GVL_1.Scope_T_Vor_WT_IN :=T_Vor_WT_IN ;
GVL_1.Scope_T_Vor_WT:=T_Vor_WT;
GVL_1.Scope_T_Vor_WT_Visu:=T_Vor_WT_Visu;
GVL_1.Scope_T_nach_WT_IN :=T_nach_WT_IN ;
GVL_1.Scope_T_nach_WT:=T_nach_WT;
GVL_1.Scope_T_nach_WT_Visu:=T_nach_WT_Visu;
GVL_1.Scope_T_HE_Einduesung_Oben_IN :=T_HE_Einduesung_Oben_IN ;
GVL_1.Scope_T_HE_Einduesung_Oben:=T_HE_Einduesung_Oben;
GVL_1.Scope_T_HE_Einduesung_Oben_Visu:=T_HE_Einduesung_Oben_Visu;
GVL_1.Scope_T_HE_Einduesung_Unten_IN :=T_HE_Einduesung_Unten_IN ;
GVL_1.Scope_T_HE_Einduesung_Unten:=T_HE_Einduesung_Unten;
GVL_1.Scope_T_HE_Einduesung_Unten_Visu:=T_HE_Einduesung_Unten_Visu;
GVL_1.Scope_T_Einduesung_Unten_IN :=T_Einduesung_Unten_IN ;
GVL_1.Scope_T_Einduesung_Unten:=T_Einduesung_Unten;
GVL_1.Scope_T_Einduesung_Unten_Visu:=T_Einduesung_Unten_Visu;
GVL_1.Scope_T_Einduesung_Oben_IN :=T_Einduesung_Oben_IN ;
GVL_1.Scope_T_Einduesung_Oben:=T_Einduesung_Oben;
GVL_1.Scope_T_Einduesung_Oben_Visu:=T_Einduesung_Oben_Visu;
GVL_1.Scope_T_Absaugung_Oben_IN :=T_Absaugung_Oben_IN ;
GVL_1.Scope_T_Absaugung_Oben:=T_Absaugung_Oben;
GVL_1.Scope_T_Absaugung_Oben_Visu:=T_Absaugung_Oben_Visu;
GVL_1.Scope_T_Absaugung_Unten_IN :=T_Absaugung_Unten_IN ;
GVL_1.Scope_T_Absaugung_Unten:=T_Absaugung_Unten;
GVL_1.Scope_T_Absaugung_Unten_Visu:=T_Absaugung_Unten_Visu;
GVL_1.Scope_T_Vor_UmdampfLuefter_IN :=T_Vor_UmdampfLuefter_IN ;
GVL_1.Scope_T_Vor_UmdampfLuefter:=T_Vor_UmdampfLuefter;
GVL_1.Scope_T_Vor_UmdampfLuefter_Visu:=T_Vor_UmdampfLuefter_Visu;
GVL_1.Scope_T_Komp_Auslass_IN :=T_Komp_Auslass_IN ;
GVL_1.Scope_T_Komp_Auslass:=T_Komp_Auslass;
GVL_1.Scope_T_Komp_Auslass_Visu:=T_Komp_Auslass_Visu;
GVL_1.Scope_T_Komp_Einlass_IN :=T_Komp_Einlass_IN ;
GVL_1.Scope_T_Komp_Einlass:=T_Komp_Einlass;
GVL_1.Scope_T_Komp_Einlass_Visu:=T_Komp_Einlass_Visu;
GVL_1.Scope_T_Kond_Auslass_IN :=T_Kond_Auslass_IN ;
GVL_1.Scope_T_Kond_Auslass:=T_Kond_Auslass;
GVL_1.Scope_T_Kond_Auslass_Visu:=T_Kond_Auslass_Visu;
GVL_1.Scope_T_DK_Oben_IN :=T_DK_Oben_IN ;
GVL_1.Scope_T_DK_Oben:=T_DK_Oben;
GVL_1.Scope_T_DK_Oben_Visu:=T_DK_Oben_Visu;
GVL_1.Scope_T_DK_Mitte_IN :=T_DK_Mitte_IN ;
GVL_1.Scope_T_DK_Mitte:=T_DK_Mitte;
GVL_1.Scope_T_DK_Mitte_Visu:=T_DK_Mitte_Visu;
GVL_1.Scope_T_DK_Unten_IN :=T_DK_Unten_IN ;
GVL_1.Scope_T_DK_Unten:=T_DK_Unten;
GVL_1.Scope_T_DK_Unten_Visu:=T_DK_Unten_Visu;
GVL_1.Scope_T_Mat_Auslass1_IN :=T_Mat_Auslass1_IN ;
GVL_1.Scope_T_Mat_Auslass1:=T_Mat_Auslass1;
GVL_1.Scope_T_Mat_Auslass1_Visu:=T_Mat_Auslass1_Visu;
GVL_1.Scope_T_Mat_Auslass2_IN :=T_Mat_Auslass2_IN ;
GVL_1.Scope_T_Mat_Auslass2:=T_Mat_Auslass2;
GVL_1.Scope_T_Mat_Auslass2_Visu:=T_Mat_Auslass2_Visu;
GVL_1.Scope_T_Mat_Auslass3_IN :=T_Mat_Auslass3_IN ;
GVL_1.Scope_T_Mat_Auslass3:=T_Mat_Auslass3;
GVL_1.Scope_T_Mat_Auslass3_Visu:=T_Mat_Auslass3_Visu;
GVL_1.Scope_T_Mat_Auslass4_IN :=T_Mat_Auslass4_IN ;
GVL_1.Scope_T_Mat_Auslass4:=T_Mat_Auslass4;
GVL_1.Scope_T_Mat_Auslass4_Visu:=T_Mat_Auslass4_Visu;
GVL_1.Scope_T_Komp_Gehaeuse_IN :=T_Komp_Gehaeuse_IN ;
GVL_1.Scope_T_Komp_Gehaeuse:=T_Komp_Gehaeuse;
GVL_1.Scope_T_Komp_Gehaeuse_Visu:=T_Komp_Gehaeuse_Visu;
GVL_1.Scope_T_DK_Band_oben1_IN :=T_DK_Band_oben1_IN ;
GVL_1.Scope_T_DK_Band_oben1:=T_DK_Band_oben1;
GVL_1.Scope_T_DK_Band_oben1_Visu:=T_DK_Band_oben1_Visu;
GVL_1.Scope_T_DK_Band_oben2_IN :=T_DK_Band_oben2_IN ;
GVL_1.Scope_T_DK_Band_oben2:=T_DK_Band_oben2;
GVL_1.Scope_T_DK_Band_oben2_Visu:=T_DK_Band_oben2_Visu;
GVL_1.Scope_T_DK_Band_oben3_IN :=T_DK_Band_oben3_IN ;
GVL_1.Scope_T_DK_Band_oben3:=T_DK_Band_oben3;
GVL_1.Scope_T_DK_Band_oben3_Visu:=T_DK_Band_oben3_Visu;
GVL_1.Scope_T_DK_Band_unten1_IN :=T_DK_Band_unten1_IN ;
GVL_1.Scope_T_DK_Band_unten1:=T_DK_Band_unten1;
GVL_1.Scope_T_DK_Band_unten1_Visu:=T_DK_Band_unten1_Visu;
GVL_1.Scope_T_DK_Band_unten2_IN :=T_DK_Band_unten2_IN ;
GVL_1.Scope_T_DK_Band_unten2:=T_DK_Band_unten2;
GVL_1.Scope_T_DK_Band_unten2_Visu:=T_DK_Band_unten2_Visu;
GVL_1.Scope_T_DK_Band_unten3_IN :=T_DK_Band_unten3_IN ;
GVL_1.Scope_T_DK_Band_unten3:=T_DK_Band_unten3;
GVL_1.Scope_T_DK_Band_unten3_Visu:=T_DK_Band_unten3_Visu;
GVL_1.Scope_T_DK_Steigband1_IN :=T_DK_Steigband1_IN ;
GVL_1.Scope_T_DK_Steigband1:=T_DK_Steigband1;
GVL_1.Scope_T_DK_Steigband1_Visu:=T_DK_Steigband1_Visu;
GVL_1.Scope_T_DK_Steigband2_IN :=T_DK_Steigband2_IN ;
GVL_1.Scope_T_DK_Steigband2:=T_DK_Steigband2;
GVL_1.Scope_T_DK_Steigband2_Visu:=T_DK_Steigband2_Visu;
GVL_1.Scope_T_DK_Steigband3_IN :=T_DK_Steigband3_IN ;
GVL_1.Scope_T_DK_Steigband3:=T_DK_Steigband3;
GVL_1.Scope_T_DK_Steigband3_Visu:=T_DK_Steigband3_Visu;
GVL_1.Scope_T_DK_Steigband4_IN :=T_DK_Steigband4_IN ;
GVL_1.Scope_T_DK_Steigband4:=T_DK_Steigband4;
GVL_1.Scope_T_DK_Steigband4_Visu:=T_DK_Steigband4_Visu;
GVL_1.Scope_Temp_Heatmatt1_IN  :=Temp_Heatmatt1_IN  ;
GVL_1.Scope_Temp_Heatmatt2_IN  :=Temp_Heatmatt2_IN  ;
GVL_1.Scope_Temp_Heatmatt3_IN  :=Temp_Heatmatt3_IN  ;
GVL_1.Scope_Temp_Heatmatt4_IN  :=Temp_Heatmatt4_IN  ;
GVL_1.Scope_Temp_Heatmatt5_IN  :=Temp_Heatmatt5_IN  ;
GVL_1.Scope_Temp_Heatmatt6_IN  :=Temp_Heatmatt6_IN  ;
GVL_1.Scope_Temp_Heatmatt7_IN  :=Temp_Heatmatt7_IN  ;
GVL_1.Scope_Temp_Heatmatt8_IN  :=Temp_Heatmatt8_IN  ;
GVL_1.Scope_Temp_Heatmatt9_IN  :=Temp_Heatmatt9_IN  ;
GVL_1.Scope_Temp_Heatmatt10_IN  :=Temp_Heatmatt10_IN  ;
GVL_1.Scope_Temp_Heatmatt1 :=Temp_Heatmatt1 ;
GVL_1.Scope_Temp_Heatmatt2 :=Temp_Heatmatt2 ;
GVL_1.Scope_Temp_Heatmatt3 :=Temp_Heatmatt3 ;
GVL_1.Scope_Temp_Heatmatt4 :=Temp_Heatmatt4 ;
GVL_1.Scope_Temp_Heatmatt5 :=Temp_Heatmatt5 ;
GVL_1.Scope_Temp_Heatmatt6 :=Temp_Heatmatt6 ;
GVL_1.Scope_Temp_Heatmatt7 :=Temp_Heatmatt7 ;
GVL_1.Scope_Temp_Heatmatt8 :=Temp_Heatmatt8 ;
GVL_1.Scope_Temp_Heatmatt9 :=Temp_Heatmatt9 ;
GVL_1.Scope_Temp_Heatmatt10 :=Temp_Heatmatt10 ;
GVL_1.Scope_Temp_compressor_Self :=Temp_compressor_Self ;
GVL_1.Scope_P_Vor_WT_IN :=P_Vor_WT_IN ;
GVL_1.Scope_P_Vor_WT:=P_Vor_WT;
GVL_1.Scope_P_Vor_WT_Visu:=P_Vor_WT_Visu;
GVL_1.Scope_P_Durchfluss_IN :=P_Durchfluss_IN ;
GVL_1.Scope_P_Durchfluss:=P_Durchfluss;
GVL_1.Scope_P_Durchfluss_Visu:=P_Durchfluss_Visu;
GVL_1.Scope_P_Komp_Einlass_IN :=P_Komp_Einlass_IN ;
GVL_1.Scope_P_Komp_Einlass:=P_Komp_Einlass;
GVL_1.Scope_P_Komp_Einlass_Visu:=P_Komp_Einlass_Visu;
GVL_1.Scope_P_Komp_Auslass_IN :=P_Komp_Auslass_IN ;
GVL_1.Scope_P_Komp_Auslass:=P_Komp_Auslass;
GVL_1.Scope_P_Komp_Auslass_Visu:=P_Komp_Auslass_Visu;
GVL_1.Scope_W_Kond_Wasser_IN :=W_Kond_Wasser_IN ;
GVL_1.Scope_W_Kond_Wasser:=W_Kond_Wasser;
GVL_1.Scope_W_Kond_Wasser_Visu:=W_Kond_Wasser_Visu;
GVL_1.Scope_O2_IN :=O2_IN ;
GVL_1.Scope_O2:=O2;
GVL_1.Scope_O2_Visu:=O2_Visu;

END_PROGRAM

// ---- POUs/FB_Blink.TcPOU
FUNCTION_BLOCK FB_Blink
VAR_INPUT
	bStart:BOOL;
	tTakt:TIME:=t#0.5s;
END_VAR
VAR_OUTPUT
	bBlink:BOOL;
END_VAR
VAR
	fbT1:TON;
	fbT2:TON;
END_VAR

(*erste Hälfte der Blinkperiode, FB-Aufruf und Beschaltung in einem *)
fbT1(IN:=bStart AND NOT fbt2.Q,
	PT:= tTakt/2,
	Q=> bBlink,
	ET=> );


(*zweite Hälfte der Blinkperiode; Bsp. programmiert mit getrennter Beschaltung und Aufruf*)

fbt2.IN := fbT1.Q;   		(*vorheriges Beschalten der InputVar*)
fbt2.PT := tTakt / 2;  	(*vorheriges Beschalten der InputVar*)

fbT2();  					(*eigentliche FB-Instanz-Aufruf*)

END_FUNCTION_BLOCK

// ---- POUs/Average.TcPOU
FUNCTION_BLOCK Average
VAR_INPUT
	Input_AV: REAL;
END_VAR
VAR_OUTPUT
	OUTPUT_AV:REAL;
END_VAR
VAR
	C_AV: INT;
	summary_AV: REAL;
END_VAR



CASE C_AV OF


0:summary_AV:=0;	C_AV:=1;
1:summary_AV:=Input_AV;	C_AV:=2;
2:summary_AV:=summary_AV+Input_AV; C_AV:=3;
3:summary_AV:=summary_AV+Input_AV; C_AV:=4;
4:summary_AV:=summary_AV+Input_AV; C_AV:=5;
5:summary_AV:=summary_AV+Input_AV; C_AV:=6;
6:summary_AV:=summary_AV+Input_AV; C_AV:=7;
7:summary_AV:=summary_AV+Input_AV; C_AV:=8;
8:summary_AV:=summary_AV+Input_AV; C_AV:=9;
9:summary_AV:=summary_AV+Input_AV; C_AV:=10;
10:summary_AV:=summary_AV+Input_AV; C_AV:=11;
11:summary_AV:=summary_AV+Input_AV; C_AV:=12;
12:summary_AV:=summary_AV+Input_AV; C_AV:=13;
13:summary_AV:=summary_AV+Input_AV; C_AV:=14;
14:summary_AV:=summary_AV+Input_AV; C_AV:=15;
15:summary_AV:=summary_AV+Input_AV; C_AV:=16;
16:summary_AV:=summary_AV+Input_AV; C_AV:=17;
17:summary_AV:=summary_AV+Input_AV; C_AV:=18;
18:summary_AV:=summary_AV+Input_AV; C_AV:=19;
19:summary_AV:=summary_AV+Input_AV; C_AV:=20;
20:summary_AV:=summary_AV+Input_AV; C_AV:=21;
21:summary_AV:=summary_AV+Input_AV; C_AV:=22;
22:summary_AV:=summary_AV+Input_AV; C_AV:=23;
23:summary_AV:=summary_AV+Input_AV; C_AV:=24;
24:summary_AV:=summary_AV+Input_AV; C_AV:=25;
25:summary_AV:=summary_AV+Input_AV; C_AV:=26;
26:summary_AV:=summary_AV+Input_AV; C_AV:=27;
27:summary_AV:=summary_AV+Input_AV; C_AV:=28;
28:summary_AV:=summary_AV+Input_AV; C_AV:=29;
29:summary_AV:=summary_AV+Input_AV; C_AV:=30;
30:summary_AV:=summary_AV+Input_AV; C_AV:=31;
31:summary_AV:=summary_AV+Input_AV; C_AV:=32;
32:summary_AV:=summary_AV+Input_AV; C_AV:=33;
33:summary_AV:=summary_AV+Input_AV; C_AV:=34;
34:summary_AV:=summary_AV+Input_AV; C_AV:=35;
35:summary_AV:=summary_AV+Input_AV; C_AV:=36;
36:summary_AV:=summary_AV+Input_AV; C_AV:=37;
37:summary_AV:=summary_AV+Input_AV; C_AV:=38;
38:summary_AV:=summary_AV+Input_AV; C_AV:=39;
39:summary_AV:=summary_AV+Input_AV; C_AV:=40;
40:summary_AV:=summary_AV+Input_AV; C_AV:=41;
41:summary_AV:=summary_AV+Input_AV; C_AV:=42;
42:summary_AV:=summary_AV+Input_AV; C_AV:=43;
43:summary_AV:=summary_AV+Input_AV; C_AV:=44;
44:summary_AV:=summary_AV+Input_AV; C_AV:=45;
45:summary_AV:=summary_AV+Input_AV; C_AV:=46;
46:summary_AV:=summary_AV+Input_AV; C_AV:=47;
47:summary_AV:=summary_AV+Input_AV; C_AV:=48;
48:summary_AV:=summary_AV+Input_AV; C_AV:=49;
49:summary_AV:=summary_AV+Input_AV; C_AV:=50;
50:summary_AV:=summary_AV+Input_AV; C_AV:=51;
51:OUTPUT_AV:=summary_AV/50.0; C_AV:=0;

END_CASE

END_FUNCTION_BLOCK

// ---- POUs/Meine_HYST.TcPOU
FUNCTION_BLOCK Meine_HYST
VAR_INPUT
	Hyst_Value: INT;
	Hyst_Low_Limit: INT;
	Hyst_Hight_Limit: INT;
END_VAR
VAR_OUTPUT
	Hyst_OUT:BOOL ;
END_VAR
VAR
(*ZEITEN*)

	TON1:TON;
	IN_T1:BOOL;
	OUT_T1:BOOL;
	TON2:TON;
	IN_T2:BOOL;
	OUT_T2:BOOL;



END_VAR




(*Hyterese Universell für Heizmatten*)

IF Hyst_Value < Hyst_Low_Limit  THEN IN_T1:=TRUE; ELSE IF Hyst_Value  >= Hyst_Hight_Limit   THEN IN_T1:=FALSE; END_IF END_IF
IF OUT_T1 THEN Hyst_OUT:=TRUE; ELSE Hyst_OUT:=FALSE; END_IF



TON1(IN:=IN_T1 , PT:=t#30s, Q=>OUT_T1 , ET=> ); (*ZEIT Hauptschütz einschalten*)

TON2(IN:=IN_T2 , PT:=t#30s, Q=>OUT_T2 , ET=> ); (*ZEIT Überwachung Hauptschütz einschalten*)

END_FUNCTION_BLOCK

// ---- POUs/Controller.TcPOU
FUNCTION_BLOCK Controller
VAR_INPUT
END_VAR
VAR_OUTPUT
END_VAR
VAR
	CTRL_1: FB_BasicPID;
	CTRL_2: FB_BasicPID;
	
	Heat_REG1_CTRL: FB_BasicPID;
	Heat_REG2_CTRL: FB_BasicPID;
	Heat_REG3_CTRL: FB_BasicPID;
	Heat_REG4_CTRL: FB_BasicPID;
	Heat_REG5_CTRL: FB_BasicPID;
	Heat_REG6_CTRL: FB_BasicPID;
	Heat_REG7_CTRL: FB_BasicPID;
	Heat_REG8_CTRL: FB_BasicPID;
	
	
	
	Heat_REG1_PWM: FB_BA_PWM;
	Heat_REG2_PWM: FB_BA_PWM;
	Heat_REG3_PWM: FB_BA_PWM;
	Heat_REG4_PWM: FB_BA_PWM;
	Heat_REG5_PWM: FB_BA_PWM;
	Heat_REG6_PWM: FB_BA_PWM;
	Heat_REG7_PWM: FB_BA_PWM;
	Heat_REG8_PWM: FB_BA_PWM;
	
	
	
	
	

END_VAR







(*Regler Kompressor*)

IF Activate_controller_comp THEN


(* Default (zurzeit nicht veränderbar)TN = 1, TV = 1,*)


CTRL_1(
	fSetpointValue:= fSollwert_comp, 
	fActualValue:=P_Komp_Auslass_Visu , 
	bReset:=Reset_Controller_comp , 
	fCtrlCycleTime:= 0.1, 
	fKp:=fKP_Controller_comp , 
	fTn:=fKI_Controller_comp , 
	fTv:=0.1 , 
	fTd:= 0.1, 
	fCtrlOutput=>fStellwert_comp , 
	nErrorStatus=>nErrorStatus_comp );
(*

VAR_INPUT
    fSetpointValue : LREAL; (* setpoint value *)
    fActualValue   : LREAL; (* actual value *)
    bReset         : BOOL;
    fCtrlCycleTime : LREAL; (* controller cycle time in seconds [s] *)
    fKp            : LREAL; (* proportional gain Kp (P) *)
    fTn            : LREAL; (* integral gain Tn (I) [s] *)
    fTv            : LREAL; (* derivative gain Tv (D-T1) [s] *)
    fTd            : LREAL; (* derivative damping time Td (D-T1) [s] *)
END_VAR
*)

ELSE

	fSollwert_comp:=0;
	fManual_controller_comp:=0;
	Set_Manual_controller_comp:=FALSE;
	fStellwert_comp:=0;

END_IF;












(* Regler 3 für Nadelregelventil*)

IF Activate_controller_Needlevalve THEN

CTRL_2(
	fSetpointValue:= fSollwert_NV, 
	fActualValue:=fRegelgroesse_NV , 
	bReset:=Reset_Controller_NV , 
	fCtrlCycleTime:= 0.1, 
	fKp:=fKP_Controller_NV , 
	fTn:=fKI_Controller_NV , 
	fTv:=0.1 , 
	fTd:= 0.1, 
	fCtrlOutput=>fStellwert_NV , 
	nErrorStatus=>nErrorStatus_NV );
	
	
(*
CTRL_3(
	ACT:=fRegelgroesse_NV,
	SET:=fSollwert_NV ,
	SUP:=0.0 ,
	OFS:= 0.0,
	M_I:= fManual_controller_NV,
	MAN:=Set_Manual_controller_NV,
	RST:= Reset_Controller_NV,
	KP:=fKP_Controller_NV,
	KI:=fKI_Controller_NV,
	LL:=0.0,
	LH:=32767 ,
	Y=>fStellwert_NV,
	DIFF=> ,
	LIM=> );
*)

ELSE


	fSollwert_NV:=0;
	 fManual_controller_NV:=0;
	Set_Manual_controller_NV:=FALSE;
	fStellwert_NV:=0;
	

END_IF;



(*Wenn Poti-Grenze Überschritten wird, wird Sollwert auf 0 gesetzt*)
IF Poti_Istwert_NV > High_Limit_Poti_Istwert_NV OR
Poti_Istwert_NV < Low_Limit_Poti_Istwert_NV THEN
Sollwert_OUT_NV:=0;
ELSE
Sollwert_OUT_NV:=REAL_TO_INT(fStellwert_NV);
END_IF;


Poti_Istwert_NV:=REAL_TO_INT(Istwert_IN_NV*100 )/32767;






(*Erklärung PID regler gemäss LIB BA*)

(*

bEn         : BOOL;
bActn       : BOOL;
bSync       : BOOL;
lrSync      : LREAL;
lrW         : LREAL;
lrX         : LREAL;
lrNZ        : LREAL;
lrYMin      : LREAL;
lrYMax      : LREAL;
lrKp        : LREAL;
udiTn       : UDINT;
udiTv       : UDINT;
udiTd       : UDINT;
udiMinToMax : UDINT;
udiMaxToMin : UDINT;
uiCycCl     : UINT;

bEn: Regleraktivierung.

bActn:Wirksinn des Reglers.

bSync / lrSync: Synchronisationsbefehl: Ausgangswert lrY auf lrSync setzen.

lrW: Sollwert.

lrX: Istwert.

lrNZ: neutrale Zone.

lrYMin: Untere Ausgabebegrenzung des Reglers.

lrYMax: Obere Ausgabebegrenzung des Reglers.

lrKp: Reglerverstärkung. Wirkt nur auf den P-Anteil.

udiTn: Nachstellzeit des I-Anteiles [ms] . Ein Nullwert an diesem Parameter schaltet den I-Anteil ab.

udiTv: Vorhaltezeit des D-Anteiles [ms] . Ein Nullwert an diesem Parameter schaltet den D-Anteil ab.

udiTd: Dämpfungszeit des D-Anteiles [ms] .

udiMinToMax: Steigungsbegrenzung des Reglerausgangs für Anstieg: udiMinToMax [s] bezogen auf eine Änderung von lrYMin auf lrYMax.

udiMaxToMin: Steigungsbegrenzung des Reglerausgangs für Abfall: udiMaxToMin [s] bezogen auf eine Änderung von lrYMax auf lrYMin.

uiCycCl: Aufrufzyklus des Bausteines als Vielfaches der Zykluszeit. Ein Nulleintrag wird automatisch als uiCycleCall=1 gewertet.
Beispiel: tTaskCycleTime = 20ms, uiCtrlCycleCall =10 -> Der Regelalgorithmus wird alle 200ms aufgerufen. Damit werden aber auch nur alle 200ms die Ausgänge aktualisiert.
VAR_OUTPUT

lrY        : LREAL;
lrE        : LREAL;
bAct       : BOOL;
b2PtAct    : BOOL;
bARW       : BOOL;
bMinLim    : BOOL;
bMaxLim    : BOOL;
bDecLim    : BOOL;
bIncLim    : BOOL;
bErr       : BOOL;
udiErrId   : UDINT;
udiErrArg  : UDINT;

lrY: Stellgröße. Bereich durch lrYMin und lrYMax eingeschränkt.

lrE: Regelabweichung (Die Berechnung ist abhängig vom Wirksinn).

bAct: Der Regler ist aktiv, das heißt freigegeben (bEn = TRUE) und nicht im Fehlerzustand (bErr = FALSE).

bARW: Anti-Reset-Windup-Funktion ist aktiv.

b2PtAct: wird nicht mehr benötigt.

bMaxLim: Die Stellgröße hat ihren oberen Grenzwert erreicht.

bMinLim: Die Stellgröße hat ihren unteren Grenzwert erreicht.

bDecLim: Die Stellgrößen-Steigung hat ihren Grenzwert für das maximale Abfallen erreicht, siehe udiMaxToMin (VAR_INPUT).

bIncLim: Die Stellgrößen-Steigung hat ihren Grenzwert für den maximale Anstieg erreicht, siehe udiMinToMax (VAR_INPUT).

bErr: Dieser Ausgang wird auf TRUE geschaltet, wenn die eingetragenen Parameter fehlerhaft sind.

udiErrId / udiErrArg: Enthält die Fehlernummer und das Fehlerargument. Siehe Fehlercodes.
*)














(*PWM Erklärung:

FB_BA_PWM

Puls-Weiten-Modulations-Baustein.

FB_BA_PWM 1:
Funktionsbeschreibung

Der Funktionsbaustein errechnet aus einem analogen Eingangssignal rIn (0..100%, intern fest begrenzt) und einer Periodendauer udiPrd [s] eine Ein- und eine Ausschaltzeit, welche an den Ausgängen als rActTiOn und rActTiOff  in Sekunden angezeigt werden.

Dabei entspricht:

    100% am Eingang einer Einschaltzeit von der gesamten Periodendauer udiPrd und einer Ausschaltzeit von 0s
    0% am Eingang einer Einschaltzeit von 0s und einer Ausschaltzeit von der gesamten Periodendauer udiPrd.

Darüber hinaus gibt es die Möglichkeit über udiMinOnTi [s] die Einschaltdauer nach unten hin zu begrenzen, um Schäden an Antrieben durch zu kurze Stellimpulse zu vermeiden. Dieses Verhalten gilt gilt jedoch nur für 0>rIn>100!
Für die Eingangssignale:

     rIn=0: Einschaltzeit=0, Ausschaltzeit=udiPrd -> bOut bleibt dauerhaft FALSE
    rIn=100: Einschaltzeit=udiPrd , Ausschaltzeit=0 -> bOut bleibt dauerhaft TRUE

Schaltverhalten

    Ein FALSE-Signal am Eingang bEn setzt den Baustein außer Funktion und bQ auf FALSE. Es werden lediglich die Ein-und Ausschaltzeiten kontinuierlich berechnet und an den Ausgängen rActTiOn und rActTiOff [s] angezeigt.
    Eine steigende Flanke am Eingang bEn aktiviert den Baustein: Er springt zunächst in einen Entscheidungs-Schritt. Je nach vorherigem Zustand vom Schaltausgang bQ wird nun in den umschaltenden Schritt gesprungen, es sei denn, der Eingang rIn steht auf 0.0. Dann erfolgt ein Sprung in den Aus-Schritt (bQ=FALSE).
    In dem jeweils aktiven Schritt (EIN oder AUS) läuft nun ein Countdown-Timer mit dem aktuell errechneten Startwert ab, der sich aus dem Puls-Pause-Verhältnis ergibt. Der Ein- bzw. Aus-Schritt wird mit der errechneten Zeit durchlaufen, egal, ob sich währenddessen das Puls-Pause-Verhältnis ändert. Der jeweilige Countdown wird an den Ausgängen udiRemTiOn und udiRemTiOff in vollen Sekunden angezeigt.
    Nach Ablauf des Ein- bzw. des Aus-Schrittes erfolgt ein Rücksprung in den Entscheidungsschritt (Punkt 2).

Ein-Ausgänge
VAR_INPUT

bEn        : BOOL;
rIn        : REAL;
udiPrd     : UDINT;
udiMinOnTi : UDINT;

bEn : Aktivierung der Puls-Weiten-Modulation.

rIn: Eingangssignal, intern auf 0..100% fest begrenzt.

udiPrd: Periodenzeit [s].

udiMinOnTi: Minimale Einschaltzeit [s].
VAR_OUTPUT

bOut        : BOOL;
bLmtSwiTi          : BOOL;
rActTiOn    : REAL;
rActTiOff   : REAL;
udiRemOnTi  : UDINT;
udiRemOffTi : UDINT;

bOut: PWM-Ausgang.

bLmtSwiTi: Informationsausgang, dass das Eingangssignal so niedrig ist, dass mit der minimalen Einschaltzeit begrenzt wird.

rActTiOn: Informationsausgang: errechnete Einschaltzeit.

rActTiOff: Informationsausgang: errechnete Ausschaltzeit.

udiRemOnTi: Countdown Einschalttimer.

udiRemOffTi: Countdown Ausschalttimer.


*)





(*PID_test(
	bEn:= , 
	bActn:= , 
	bSync:= , 
	lrSync:= , 
	lrW:= , 
	lrX:= , 
	lrNz:= , 
	lrYMin:= , 
	lrYMax:= , 
	lrKp:= , 
	udiTn:= , 
	udiTv:= , 
	udiTd:= , 
	udiMinToMax:= , 
	udiMaxToMin:= , 
	uiCycCl:= , 
	lrY=> , 
	lrE=> , 
	bAct=> , 
	b2PtAct=> , 
	bARW=> , 
	bMinLim=> , 
	bMaxLim=> , 
	bDecLim=> , 
	bIncLim=> , 
	bErr=> , 
	udiErrId=> , 
	udiErrArg=> );*)

	
	
//Verknüpfung = PID Regler => PWM => OUTPUT
	
//Heizregister Gruppe 1 oben 1-4

Heat_REG1_CTRL(
	fSetpointValue:= fSetpointValue1, 
	fActualValue:=fTemp_mean_belt_top, 
	bReset:=Reset_heatreg_top, 
	fCtrlCycleTime:= 0.1, 
	fKp:=fKP_Controller_Heatmatt1 , 
	fTn:=fKI_Controller_Heatmatt1 , 
	fTv:=0.1 , 
	fTd:= 0.1, 
	fCtrlOutput=>fPWMDutyCycle1, 
	nErrorStatus=>nErrorStatus_Heatmatt1 );
	
	//
	
	Heat_REG1_PWM(
	bEn:=TRUE , 
	rIn:= fPWMDutyCycle1	, 
	udiPrd:=2, //2 =sekunde
	udiMinOnTi:=1 , //1 =sekunde
	bQ=>bAuto_Heat_REG1_CTRL, 
	bLmtMinOnTi=> , 
	rActTiOn=> , 
	rActTiOff=> , 
	udiRemTiOn=> , 
	udiRemTiOff=> );
	
	
	
	
	
	
	
	
	//Heizregister Gruppe 2 unten 5-8

	
	Heat_REG2_CTRL(	
	fSetpointValue:= fSetpointValue2, 
	fActualValue:=fTemp_mean_belt_bottom, 
	bReset:=Reset_heatreg_bottom , 
	fCtrlCycleTime:= 0.1, 
	fKp:=fKP_Controller_Heatmatt2 , 
	fTn:=fKI_Controller_Heatmatt2 , 
	fTv:=0.1 , 
	fTd:= 0.1, 
	fCtrlOutput=>fPWMDutyCycle2, 
	nErrorStatus=>nErrorStatus_Heatmatt2 );

	Heat_REG2_PWM(
	bEn:=TRUE , 
	rIn:= fPWMDutyCycle2	, 
	udiPrd:=2, //2 =sekunde
	udiMinOnTi:=1 , //1 =sekunde
	bQ=>bAuto_Heat_REG2_CTRL, 
	bLmtMinOnTi=> , 
	rActTiOn=> , 
	rActTiOff=> , 
	udiRemTiOn=> , 
	udiRemTiOff=> );
	
	
	
//Heizregister bei Kompressor (verhinderung von Kondensation)
	
Heat_REG3_CTRL(	
	fSetpointValue:= fSetpointValue3, 
	fActualValue:= Temp_Heatmatt3 , 
	bReset:= Reset_heatreg_compressor, 
	fCtrlCycleTime:= 0.1, 
	fKp:=fKP_Controller_Heatmatt3 , 
	fTn:=fKI_Controller_Heatmatt3 , 
	fTv:=0.1 , 
	fTd:= 0.1, 
	fCtrlOutput=>fPWMDutyCycle3, 
	nErrorStatus=>nErrorStatus_Heatmatt3 );


	Heat_REG3_PWM(
	bEn:=TRUE , 
	rIn:= fPWMDutyCycle3	, 
	udiPrd:=2, //2 =sekunde
	udiMinOnTi:=1 , //1 =sekunde
	bQ=>bAuto_Heat_REG3_CTRL, 
	bLmtMinOnTi=> , 
	rActTiOn=> , 
	rActTiOff=> , 
	udiRemTiOn=> , 
	udiRemTiOff=> );
	
	
	
(* REserve*)	

(*
Heat_REG4_CTRL(	
	fSetpointValue:= fSetpointValue4, 
	fActualValue:= Temp_Heatmatt4 , 
	bReset:= , 
	fCtrlCycleTime:= 0.1, 
	fKp:=fKP_Controller_Heatmatt4 , 
	fTn:=fKI_Controller_Heatmatt4 , 
	fTv:=0.1 , 
	fTd:= 0.1, 
	fCtrlOutput=>fPWMDutyCycle4, 
	nErrorStatus=>nErrorStatus_Heatmatt4 );

	*)
	


(* Der Regler soll vorübergehend so funktionieren, dass im Haupt-Manu Mode der regeler im Auto-Modus läuft*)
	IF Ctr_Manu AND Control_Manu_active =FALSE THEN

	 Ctr_Manu_active:=TRUE;
	 Ctr_Auto_active:=FALSE;
	 Ctr_Reset_active:=FALSE;
	ELSE IF Control_Manu_active THEN
	
	 Ctr_Manu_active:=FALSE;
	 Ctr_Auto_active:=TRUE;
	 Ctr_Reset_active:=FALSE;
	ELSE IF Ctr_Reset THEN
	 Ctr_Manu_active:=FALSE;
	 Ctr_Auto_active:=FALSE;
	 Ctr_Reset_active:=TRUE;
	
	END_IF
	END_IF
	END_IF



	
	

(*Wichtige info: Zurzeit  ist der Manu-Ausgang der Haupt-Ausgang, auch wenn der Regler im Auto_Modus arbeitet*)



//Regler Heizregister 1-4 und 5-8

IF T_HE_Einduesung_Oben_Visu > T_Limit_Heatreg_top  OR 
fTemp_mean_belt_top > T_Limit_Heatreg_top OR
OK_For_HEAT_WHILE_FAN_IS_ON = FALSE THEN
HEAT_Reg_1_Manu:=FALSE;
bAuto_Heat_REG1_CTRL:=FALSE;
ELSE
HEAT_Reg_1_Manu:=bManuHeat_REG1_CTRL OR bAuto_Heat_REG1_CTRL;
END_IF;

IF T_HE_Einduesung_unten_Visu > T_Limit_Heatreg_bottom  OR 
fTemp_mean_belt_bottom > T_Limit_Heatreg_bottom OR
OK_For_HEAT_WHILE_FAN_IS_ON = FALSE THEN
HEAT_Reg_2_Manu:=FALSE;
bAuto_Heat_REG2_CTRL:=FALSE;
ELSE
HEAT_Reg_2_Manu:=bManuHeat_REG2_CTRL OR bAuto_Heat_REG2_CTRL;
END_IF;



//OK_For_HEAT_WHILE_FAN_IS_ON:=SteamFAN_Switch_ON_manu AND SteamFan_ON_manu AND Setpoint_SteamFan_Visu >=0;

//Versuch mal so, wiel Preobleme mit Zeile oben:
IF SteamFAN_Switch_ON_manu AND SteamFan_ON_manu AND Setpoint_SteamFan_Visu > 0 THEN
OK_For_HEAT_WHILE_FAN_IS_ON:=TRUE;
ELSE
OK_For_HEAT_WHILE_FAN_IS_ON:=FALSE;
END_IF;

//Heizregister bei Kompressor (verhinderung von Kondensation)


IF T_Monitor_Heatreg1 > T_Limit_Heatreg  OR T_Monitor_Heatreg2 > T_Limit_Heatreg THEN

HEAT_Reg_3_Manu:=FALSE;
//HEAT_Reg_4_Manu:=FALSE;
ELSE
	
HEAT_Reg_3_Manu:=bManuHeat_REG3_CTRL OR bAuto_Heat_REG3_CTRL;
//HEAT_Reg_4_Manu:=bManuHeat_REG4_CTRL OR bAuto_Heat_REG4_CTRL;

END_IF;






	(*Hier wird der Setpoint automatisch auf 0 gesetzt*)



	IF  Main_Relais = FALSE THEN
		
	bManuHeat_REG1_CTRL:=FALSE;
	bManuHeat_REG2_CTRL:=FALSE;
	bManuHeat_REG3_CTRL:=FALSE;
	bManuHeat_REG4_CTRL:=FALSE;
	
	bAuto_Heat_REG1_CTRL:=FALSE;
	bAuto_Heat_REG2_CTRL:=FALSE;
	bAuto_Heat_REG3_CTRL:=FALSE;
	bAuto_Heat_REG4_CTRL:=FALSE;
	
	fSetpointValue1:=0;
	fSetpointValue2:=0;
	fSetpointValue3:=0;
	fSetpointValue4:=0;
	
	
	END_IF;








fTemp_mean_belt_top:= (T_DK_Band_oben1_Visu + T_DK_Band_oben3_Visu) /2.0;

fTemp_mean_belt_bottom:= (T_DK_Band_unten1_Visu+ T_DK_Band_unten3_Visu) /2.0;

END_FUNCTION_BLOCK

// ---- POUs/FB_PeerToPeer.TcPOU
(* Function block example of UDP peer-to-peer application *)
FUNCTION_BLOCK FB_PeerToPeer
VAR_IN_OUT
	fbTx		: FB_FrameFifo;(* TX fifo *)
	fbRx		: FB_FrameFifo;(* RX fifo *)
	fbLog		: FB_LogFifo;(* Log message fifo *)
END_VAR
VAR_INPUT
	sSrvNetId		: T_AmsNetID 	:= '';(* TwinCAT TCP/IP server network address. Default: empty string. *)
	sLocalHost		: T_IPv4Addr 	:= '192.168.100.88';(* Local address: String containing an (Ipv4) Internet Protocol dotted address. *)
	nLocalPort		: UDINT 		:= 0;(* Local address: IP port number. *)
	bEnable 		: BOOL			:= true;(* TRUE => Enable/connect, FALSE => Disable/disconnect *)
	tReconnect		: TIME			:= T#5S;(* Reconnect delay time *)
	bLog			: BOOL			:= FALSE;(* TRUE => Enable log message output, FALSE => Disable *)
	sPrefix			: STRING 		:= 'PeerToPeerX::';(* Log message description string (allows the identification of log message source) *)
END_VAR
VAR_OUTPUT
	bCreated		: BOOL;(* Connectionless socket state (TRUE => created, FALSE => closed) *)
END_VAR
VAR
	fbCreate		: FB_SocketUdpCreate;
	fbClose			: FB_SocketClose;
	fbReceiveFrom	: FB_SocketUdpReceiveFrom;
	fbSendTo		: FB_SocketUdpSendTo;
	stSendTo		: ST_FrameFifoEntry;
	stReceivedFrom	: ST_FrameFifoEntry;
	fbCreateTimer	: TON := ( PT := T#0S );	
	eStep			: E_ClientServerSteps;
END_VAR



//für ehemals test mit IAS kann die UPD kommunikation verwendet werden!


(*

CASE eStep OF
	eUDP_STATE_IDLE:
		IF bEnable XOR bCreated THEN
			IF bEnable THEN
				fbTx.Clear( sPrefix := CONCAT( sPrefix, 'FB_FrameFifo(sender)::' ), bLog := bLog );(* Clear send fifo *)
				fbRx.Clear( sPrefix := CONCAT( sPrefix, 'FB_FrameFifo(receiver)::' ), bLog := bLog );(* Clear receiver fifo *)
				fbLog.Clear( sPrefix := sPrefix, bLog := bLog );(* Clear log fifo *)

				(* At program start (first time) connect emmediately, next time after delay time *)
				fbCreateTimer( IN := TRUE );
				IF fbCreateTimer.Q THEN
					fbCreateTimer( IN := FALSE, PT := tReconnect ); 
					eStep := eUDP_STATE_CREATE_START;
				END_IF
			
			ELSE
				eStep := eUDP_STATE_CLOSE_START;
			END_IF
		ELSIF bCreated THEN
			fbTx.RemoveHead( stGet => stSendTo );
			IF fbTx.bOk THEN
				eStep := eUDP_STATE_SEND_START;
			ELSE (* Empty *)
				eStep := eUDP_STATE_RECEIVE_START;
			END_IF
		ELSE
			fbCreateTimer( IN := FALSE, PT := T#0S );
		END_IF

	eUDP_STATE_CREATE_START:
		fbCreate( bExecute := FALSE  );
		fbCreate( sSrvNetId := sSrvNetId, sLocalHost:= sLocalHost, nLocalPort:= nLocalPort, bExecute:= TRUE );
		eStep := eUDP_STATE_CREATE_WAIT;

	eUDP_STATE_CREATE_WAIT:
		fbCreate( bExecute := FALSE );
		IF NOT fbCreate.bBusy THEN
			IF NOT fbCreate.bError THEN
				bCreated := TRUE;
				fbLog.Message( sMessage := 'Connectionless (UDP) socket created!', hSocket := fbCreate.hSocket );
				eStep := eUDP_STATE_IDLE;
			ELSE
				fbLog.Error( sMessage := 'FB_SocketUdpCreate()', nErrID := fbCreate.nErrID );
				eStep := eUDP_STATE_ERROR;
			END_IF
		END_IF

	eUDP_STATE_SEND_START:
		fbSendTo( bExecute := FALSE );
		fbSendTo( sSrvNetId := sSrvNetId, sRemoteHost := stSendTo.stRemoteAddr.sAddr,
					nRemotePort := stSendTo.stRemoteAddr.nPort,
					pSrc:= ADR( stSendTo.sMessage ),
					cbLen:= INT_TO_UDINT(LEN( stSendTo.sMessage )) + 1, (* Include the end delimiter *)
					hSocket:= fbCreate.hSocket, bExecute:= TRUE );
		eStep := eUDP_STATE_SEND_WAIT;

	eUDP_STATE_SEND_WAIT:
		fbSendTo( bExecute := FALSE );
		IF NOT fbSendTo.bBusy THEN
			IF NOT fbSendTo.bError THEN
				eStep := eUDP_STATE_RECEIVE_START;
			ELSE
				fbLog.Error( sMessage := 'FB_SocketUdpSendTo()', nErrID := fbSendTo.nErrID );
				eStep := eUDP_STATE_ERROR;
			END_IF
		END_IF

	eUDP_STATE_RECEIVE_START:
		MEMSET( ADR( stReceivedFrom ), 0, SIZEOF( stReceivedFrom ) );
		fbReceiveFrom( bExecute := FALSE );
		fbReceiveFrom( sSrvNetId := sSrvNetId, 
						pDest:= ADR( stReceivedFrom.sMessage ),
						cbLen:= SIZEOF( stReceivedFrom.sMessage ) - 1, (* Without string delimiter *)
						hSocket:= fbCreate.hSocket, bExecute:= TRUE );
		eStep := eUDP_STATE_RECEIVE_WAIT;

	eUDP_STATE_RECEIVE_WAIT:
		fbReceiveFrom( bExecute := FALSE );
		IF NOT fbReceiveFrom.bBusy THEN
			IF NOT fbReceiveFrom.bError THEN
				IF fbReceiveFrom.nRecBytes > 0 THEN
					
					stReceivedFrom.stRemoteAddr.sAddr := fbReceiveFrom.sRemoteHost;
					stReceivedFrom.stRemoteAddr.nPort := fbReceiveFrom.nRemotePort;
					
					fbRx.AddTail( stPut := stReceivedFrom );
					IF NOT fbRx.bOk THEN(* Check for fifo overflow *)
						fbLog.Error( sMessage :='FB_FrameFifo(receiver)', nErrID := PLCPRJ_ERROR_RECFIFO_OVERFLOW );
					END_IF
				END_IF
				eStep := eUDP_STATE_IDLE;
			ELSE
				fbLog.Error( sMessage := 'FB_SocketUdpReceiveFrom()', nErrID := fbReceiveFrom.nErrID );
				IF fbReceiveFrom.nErrID = 16#80072746 THEN(* Connection is reset by remote side *)
					eStep := eUDP_STATE_IDLE;
				ELSE
					eStep := eUDP_STATE_ERROR;
				END_IF
			END_IF
		END_IF

	eUDP_STATE_CLOSE_START:
		fbLog.Message( sMessage := 'Closing connectionless (UDP) socket!', hSocket := fbCreate.hSocket );
		fbClose( bExecute := FALSE );
		fbClose( sSrvNetId := sSrvNetId, hSocket := fbCreate.hSocket, bExecute := TRUE );
		eStep := eUDP_STATE_CLOSE_WAIT;

	eUDP_STATE_CLOSE_WAIT:
		fbClose( bExecute := FALSE );
		IF NOT fbClose.bBusy THEN
			bCreated := FALSE;
			IF NOT fbClose.bError THEN
				eStep := eUDP_STATE_IDLE;
			ELSE
				fbLog.Error( sMessage := 'FB_SocketClose()', nErrID := fbClose.nErrID );
				eStep := eUDP_STATE_ERROR;
			END_IF
		END_IF

	eUDP_STATE_ERROR: (* Error step *)
		IF bCreated THEN
			eStep := eUDP_STATE_CLOSE_START;
		ELSE
			eStep := eUDP_STATE_IDLE;
		END_IF
END_CASE
*)

END_FUNCTION_BLOCK

// ---- POUs/Helper POUs/FB_FrameFifo.TcPOU
(* Tx/Rx (string data) fifo control function block *)
FUNCTION_BLOCK FB_FrameFifo
VAR_INPUT
	bLog		: BOOL := FALSE;(* TRUE => Enable log message output, FALSE => Disable *)
	sPrefix		: STRING := 'Unknown::';(* Log message description string (allows the identification of log message source) *)
	stPut		: ST_FrameFifoEntry;(* Frame entry to add (write) to the buffer *)
END_VAR
VAR_OUTPUT
	bOk			: BOOL;(* TRUE = New entry added or removed succesfully, FALSE = Fifo overflow or fifo empty *)
	stGet		: ST_FrameFifoEntry;(* Frame entry removed (read) from fifo *)
	nCount		: UDINT := 0;(* Number of fifo entries *)
END_VAR
VAR
	fbBuffer 	: FB_MemRingBuffer;(* Basic (lower level) string buffer control function block *)
	buffer		: ARRAY[0..PLCPRJ_BUFFER_SIZE] OF BYTE;(* Internal buffer memory *)
END_VAR

;

ACTION AddTail:
(* Adds new fifo entry *)
fbBuffer.A_AddTail( pBuffer:= ADR(buffer), cbBuffer:= SIZEOF(buffer),
					pWrite:= ADR( stPut ), cbWrite := SIZEOF( stPut ), 
					bOk=>bOk, nCount=>nCount );
IF bOk AND bLog THEN(* Log message *)
	ADSLOGSTR( ADSLOG_MSGTYPE_HINT OR ADSLOG_MSGTYPE_LOG, 
			CONCAT( CONCAT( sPrefix, SOCKETADDR_TO_STRING(stPut.stRemoteAddr) ), '>>"%s"' ),
			stPut.sMessage );
END_IF
END_ACTION

ACTION Clear:
(* Clears all fifo entries *)
stGet.sMessage := '';
stGet.stRemoteAddr.nPort := 0;
stGet.stRemoteAddr.sAddr := '';
fbBuffer.A_Reset( pBuffer := ADR( buffer ), cbBuffer := SIZEOF( buffer ), 
					bOk=>bOk, nCount=>nCount );
END_ACTION

ACTION RemoveHead:
(* Removes oldest fifo entry *)
IF nCount = 0 THEN
	stGet.sMessage := '';
	stGet.stRemoteAddr.nPort := 0;
	stGet.stRemoteAddr.sAddr := '';
	bOk := FALSE;
	RETURN;
END_IF

fbBuffer.A_RemoveHead( pBuffer:= ADR(buffer), cbBuffer:= SIZEOF(buffer),
						pRead := ADR( stGet ), cbRead := SIZEOF( stGet ),
						bOk=>bOk, nCount=>nCount );
END_ACTION

END_FUNCTION_BLOCK

// ---- POUs/Helper POUs/FB_LogFifo.TcPOU
(* Log/debug/error message fifo *)
FUNCTION_BLOCK FB_LogFifo
VAR_INPUT
	bLog		: BOOL 		:= FALSE;(* TRUE => Enable log message output, FALSE => Disable *)
	sPrefix		: STRING 	:= 'Unknown::';(* Log message description string (allows the identification of log message source) *)
	
	sMessage	: STRING 	:= '';(* String message to add (write) to the fifo *)
	nErrID		: UDINT 	:= 0;(* Error code to add (write) to the fifo *)
	hSocket		: T_HSOCKET;(* Socket connection handle *)
END_VAR
VAR_OUTPUT
	bOk			: BOOL;(* TRUE = New entry added or removed succesfully, FALSE = Fifo overflow or fifo empty *)
	sGet		: T_MaxString := '';(* String entry removed (read) from fifo *)
	nCount		: UDINT := 0;(* Number of fifo entries *)
END_VAR
VAR
	fbBuffer 	: FB_StringRingBuffer;(* Basic (lower level) string buffer control function block *)
	buffer		: ARRAY[0..PLCPRJ_BUFFER_SIZE] OF BYTE;(* Internal buffer memory *)
	sSource		: T_MaxString;	
	sPut		: T_MaxString;
END_VAR

;

ACTION Clear:
(* Clears all fifo entries *)
fbBuffer.A_Reset( 	pBuffer := ADR( buffer ), cbBuffer := SIZEOF( buffer ), 
					bOk=>bOk, nCount=>nCount, getValue=>sGet );
END_ACTION

ACTION Error:
(* Adds new fifo entry *)
IF nErrID = 0 THEN
	sSource := '::Error: 0x';
ELSIF ( nErrID AND 16#80000000) = 16#80000000 THEN
	IF nErrID = 16#80072746 THEN
		sSource := '::Win32 error (the connection is reset by remote side): 0x';
	ELSE
		sSource := '::Win32 error: 0x';
	END_IF
ELSIF (nErrID AND 16#00008100) = 16#00008100 THEN
	CASE nErrID OF
		PLCPRJ_ERROR_SENDFIFO_OVERFLOW:
			sSource := '::PLC sample project send fifo overflow error: 0x';
		PLCPRJ_ERROR_RECFIFO_OVERFLOW:
			sSource := '::PLC sample project receive fifo overflow error: 0x';
	ELSE
		sSource := '::Other PLC sample project error: 0x';
	END_CASE
ELSIF (nErrID AND 16#00008000) = 16#00008000 THEN
	sSource := '::Internal TCP/IP Connection Server error: 0x';
ELSE
	sSource := '::TwinCAT System error: 0x';
END_IF

sPut := CONCAT( CONCAT( CONCAT( sPrefix, sMessage ), sSource ), DWORD_TO_HEXSTR( nErrID AND 16#FFFF, 0, FALSE ) ); 

fbBuffer.A_AddTail( pBuffer:= ADR(buffer), cbBuffer:= SIZEOF(buffer),
					putValue:= sPut, bOk=>bOk, nCount=>nCount );
IF bOk THEN
	IF bLog THEN(* Log error message *)
		ADSLOGSTR( ADSLOG_MSGTYPE_ERROR OR ADSLOG_MSGTYPE_LOG, '%s', sPut );	
	END_IF
END_IF
END_ACTION

ACTION Message:
(* Adds new fifo entry *)
sPut := CONCAT( CONCAT( sPrefix, sMessage ), CONCAT( '::', SOCKETADDR_TO_STRING(hSocket.localAddr) ) );
fbBuffer.A_AddTail( pBuffer:= ADR(buffer), cbBuffer:= SIZEOF(buffer),
					putValue:= sPut, bOk=>bOk, nCount=>nCount );
IF bOk THEN
	IF bLog THEN(* Log information message *)
		ADSLOGSTR( ADSLOG_MSGTYPE_HINT OR ADSLOG_MSGTYPE_LOG, '%s', sPut );	
	END_IF
END_IF
END_ACTION

ACTION Remove:
(* Removes oldest fifo entry *)
IF nCount = 0 THEN
	sGet := '';
	bOk := FALSE;
	RETURN;
END_IF

fbBuffer.A_RemoveHead( pBuffer:= ADR(buffer), cbBuffer:= SIZEOF(buffer),
						getValue=>sGet, bOk=>bOk, nCount=>nCount );
END_ACTION

END_FUNCTION_BLOCK

// ---- GlobalTextList.TcGTLO
TEXTLIST GlobalTextList
  81 = '% s'
  184 = '%2.1f %'
  220 = '%2.1f (mbar)'
  188 = '%2.1f KI (%)'
  187 = '%2.1f KP (%)'
  124 = '%2.1f Value Comp PT100'
  36 = '%2u'
  32 = '%2u '
  185 = '%2u %'
  91 = '%3.2f'
  103 = '%3.2f  '
  152 = '%3.2f  (mbar)'
  50 = '%3.2f  (°C)'
  217 = '%3.2f  Heizband2'
  218 = '%3.2f  Heizband3'
  141 = '%3.2f  SEO2 1.51'
  122 = '%3.2f  SEP1.11'
  119 = '%3.2f  SEP2.11'
  121 = '%3.2f  SEP2.12'
  90 = '%3.2f  SET2.8'
  227 = '%3.2f  SET3.8'
  142 = '%3.2f  SEW 2.31'
  219 = '%3.2f  T.Mittel'
  205 = '%3.2f (ms)'
  149 = '%3.2f Comp.L1'
  150 = '%3.2f Comp.L2'
  151 = '%3.2f Comp.L3'
  99 = '%3.2f Heatreg 2'
  100 = '%3.2f Heatreg1'
  128 = '%3.2f Heatreg2'
  101 = '%3.2f Heatreg3'
  157 = '%3.2f Heatreg4'
  158 = '%3.2f Heatreg5'
  159 = '%3.2f Heatreg6'
  160 = '%3.2f Heatreg7'
  161 = '%3.2f Heatreg8'
  146 = '%3.2f Main L1'
  147 = '%3.2f Main L2'
  148 = '%3.2f Main L3'
  109 = '%3.2f SET 1.01'
  110 = '%3.2f SET 1.02 '
  111 = '%3.2f SET 1.03 '
  112 = '%3.2f SET 1.04 '
  113 = '%3.2f SET 1.05'
  114 = '%3.2f SET 1.06'
  115 = '%3.2f SET 1.07'
  116 = '%3.2f SET 1.08'
  117 = '%3.2f SET 1.09'
  173 = '%3.2f SET 1.81 '
  174 = '%3.2f SET 1.82'
  175 = '%3.2f SET 1.83'
  176 = '%3.2f SET 1.91'
  177 = '%3.2f SET 1.92'
  178 = '%3.2f SET 1.93'
  162 = '%3.2f SET 2.01'
  163 = '%3.2f SET 2.02 '
  164 = '%3.2f SET 2.03 '
  165 = '%3.2f SET 3.01 '
  166 = '%3.2f SET 3.02'
  167 = '%3.2f SET 3.03'
  168 = '%3.2f SET 3.71'
  169 = '%3.2f SET 3.72'
  170 = '%3.2f SET 3.73'
  171 = '%3.2f SET 3.74'
  2317 = '%3.2f SET 3.75'
  738 = '%3.2f SET 3.76'
  553 = '%3.2f SET 3.77'
  2540 = '%3.2f SET 3.78'
  179 = '%3.2f SET 3.81'
  180 = '%3.2f SET 3.82'
  181 = '%3.2f SET 3.83'
  182 = '%3.2f SET 3.84'
  2060 = '%3.2f SET 3.85'
  607 = '%3.2f SET 3.86'
  2031 = '%3.2f SET 3.87'
  1483 = '%3.2f SET 3.88'
  172 = '%3.2f SET 4.01'
  140 = '%3.2f SET Ambiente'
  236 = '%3.2f Tauch-HZ. L1'
  235 = '%3.2f Tauch-HZ. L2'
  234 = '%3.2f Tauch-HZ. L3'
  125 = '%3.2f UD  L1'
  126 = '%3.2f UD  L2'
  127 = '%3.2f UD  L3'
  130 = '%3u Temp. Heatmatt1 '
  139 = '%3u Temp. Heatmatt10 '
  131 = '%3u Temp. Heatmatt2 '
  132 = '%3u Temp. Heatmatt3 '
  133 = '%3u Temp. Heatmatt4 '
  134 = '%3u Temp. Heatmatt5 '
  135 = '%3u Temp. Heatmatt6 '
  136 = '%3u Temp. Heatmatt7 '
  137 = '%3u Temp. Heatmatt8'
  138 = '%3u Temp. Heatmatt9 '
  24 = '%s'
  191 = 'Activate'
  20 = 'Advanced\nControl'
  186 = 'Ausgabe Stellwert'
  17 = 'Auto'
  87 = 'Auto active'
  92 = 'Auto-Output'
  1577 = 'Back'
  1699 = 'back'
  28 = 'Check Comp\nTemperature!'
  257 = 'Close HMI'
  27 = 'Continue\nStartup'
  68 = 'Current Total [A]'
  86 = 'Default=Auto active'
  216 = 'DO1'
  230 = 'DO2'
  233 = 'DO3'
  231 = 'DO4'
  120 = 'Druck (mBar):'
  25 = 'Durchmesser in mm eingeben'
  98 = 'Duty Cycle'
  69 = 'Electrical Power [kW]'
  344 = 'forward'
  40 = 'FU OK'
  38 = 'FU ON'
  13 = 'Group1'
  12 = 'Group2'
  11 = 'Group3'
  97 = 'Hauptschütz'
  2425 = 'Heat \nController'
  250 = 'Heat Controller'
  155 = 'Heatregister'
  226 = 'Heizeinschraubkörper:'
  74 = 'Heizelemente ON/OFF'
  10 = 'Heizmatten'
  73 = 'Heizmatten ON/OFF'
  143 = 'Heizmatten:'
  215 = 'Heizregister Kompressor'
  89 = 'Heizregister:'
  85 = 'Heizreglerbetrieb:'
  43 = 'Hysterese hoch (°C)'
  42 = 'Hysterese tief (°C)'
  210 = 'In Progress'
  223 = 'Integralwert'
  225 = 'Istwert Vordruck Scrolli'
  154 = 'Kompressor'
  153 = 'Kompressoreinlass'
  228 = 'L1:'
  229 = 'L2:'
  232 = 'L3:'
  2114 = 'Layout'
  752 = 'Main'
  14 = 'Main ON'
  94 = 'Main-Output'
  129 = 'Main: in (A)'
  19 = 'Manu'
  93 = 'Manu-Output'
  34 = 'MANUEL BETRIEB'
  955 = 'MANUELBETRIEB'
  0 = 'Mat1'
  9 = 'Mat10'
  2 = 'Mat2'
  4 = 'Mat3'
  6 = 'Mat4'
  8 = 'Mat5'
  1 = 'Mat6'
  3 = 'Mat7'
  5 = 'Mat8'
  7 = 'Mat9'
  207 = 'Next Step'
  29 = 'OK for \nOperation'
  88 = 'ON/OFF'
  23 = 'ON1'
  22 = 'ON2'
  21 = 'ON3'
  368 = 'PID'
  71 = 'Press. Umg'
  224 = 'Proportionalwert'
  33 = 'PWM Output 0-100%'
  96 = 'Ref. Temp'
  903 = 'Regelparameter Heizreister oben'
  183 = 'Regelparameter Kompressor Klauenkolben'
  193 = 'Regelparameter Kompressor Scrolli'
  192 = 'Regelparameter Nadelventil'
  61 = 'Rel. P OUT'
  62 = 'Rel. P TM'
  54 = 'Rel. P WT'
  18 = 'Reset'
  15 = 'Reset '
  213 = 'Reset Seq.'
  67 = 'RPM Des. Venti [%]'
  65 = 'RPM Kompressor [%]'
  238 = 'S'
  209 = 'Schrittnummer:'
  37 = 'Schütz'
  59 = 'SE-P2.2'
  56 = 'SE-P2.5'
  64 = 'SE-P3.11'
  57 = 'SE-P3.3'
  76 = 'SE-P3.32'
  63 = 'SE-P6.2'
  60 = 'SE-T2.3'
  78 = 'SE-T2.51'
  80 = 'SE-T2.52'
  55 = 'SE-T2.6'
  53 = 'SE-T2.8'
  70 = 'SE-T3.31'
  77 = 'SE-T3.33'
  58 = 'SE-T3.4'
  66 = 'SE-T3.51'
  79 = 'SE-T3.52'
  869 = 'Send Trigger'
  241 = 'Sensors'
  212 = 'Sequence End'
  2084 = 'Service'
  2578 = 'Service2'
  95 = 'Setpoint'
  242 = 'Show'
  123 = 'Sicherheitstemps:'
  239 = 'Sollwert'
  190 = 'Sollwert Druck Dampfkammer'
  49 = 'Sollwert Horizontalband'
  39 = 'Sollwert Kompressor'
  222 = 'Sollwert Primär Kompressor'
  52 = 'Sollwert Steigförderer'
  370 = 'Sollwert Umdampfventi'
  35 = 'Sollwert Umdampfventilator'
  221 = 'Sollwert Vordruck Scrolli'
  26 = 'Start\nAutostart'
  208 = 'Start Again'
  211 = 'Start Point'
  30 = 'Startup\nfinished'
  31 = 'Startup Active'
  1383 = 'Steamfan OK'
  657 = 'Steamfan OK\nfor heating'
  1676 = 'Steamfan OK\nfot heating'
  189 = 'Stellwert Kompressor Manu'
  214 = 'Step back'
  102 = 'Stromverbrauch: in (A)'
  16 = 'Switch OFF'
  627 = 'Switch OFF\t'
  1043 = 'T.Monitor '
  105 = 'T.Monitor 1 SE-T 1.03'
  107 = 'T.Monitor 1 SE-T 1.04'
  106 = 'T.Monitor 2 SE-T 1.05'
  108 = 'T.Monitor 2 SE-T 1.06'
  2391 = 'T.Monitor Mean Values'
  2101 = 'T.Monitor Mean Values  '
  2587 = 'T.Monitor xy'
  41 = 'Temp\nError'
  145 = 'Temp\nError comp.'
  144 = 'Temp\nError SteamFan'
  1489 = 'Temp. \nKompressor \nGehause'
  237 = 'Temp. \nKompressor Gehause'
  51 = 'Temp. Kompressor Gehause'
  72 = 'Temp. Umg'
  118 = 'Temperaturen (°C):'
  104 = 'Tempimit switch OFF (°C)\ngroup TOP'
  1589 = 'Testseite'
  75 = 'TM'
  2371 = 'UDP-Kommunikation'
  156 = 'Umdampfventi'
  240 = 'V Main'
  203 = 'V-Dichtring\nAuslass'
  202 = 'V-Dichtring\nEinlass'
  47 = 'V1'
  44 = 'V2'
  45 = 'V3'
  46 = 'V4'
  48 = 'V5'
  1447 = 'V6'
  196 = 'Vacuum1'
  195 = 'Vacuum2'
  1501 = 'VE-K 2.71\n\n\nVE-K 2.72\n\n\nVE-K 2.73'
  829 = 'VE-K 2.71\n\nVE-K 2.72\n\nVE-K 2.73'
  84 = 'VE-K 2.71\n\nVE-K 2.73'
  82 = 'VE-K2.71'
  511 = 'VE-K2.72'
  83 = 'VE-K2.73'
  194 = 'VE-K3.05'
  197 = 'VE-K3.06'
  198 = 'VE-K3.13'
  199 = 'VE-K3.19'
  200 = 'VE-K3.20'
  201 = 'VE-K3.21'
  204 = 'VE-K3.22'
  206 = 'Zykluszeit Reglerausgnag (ms)'
END_TEXTLIST
